// TIA Portal V20 program export: 0 tag tables, 0 data types, 0 data blocks, 4 code blocks (in call order from the OBs), 0 instance data blocks

ORGANIZATION_BLOCK "Main"   // OB1, LAD, ProgramCycle
TITLE = "Main Program Sweep (Cycle)"
{ S7_Optimized_Access := 'TRUE' }
// stored: SetENOAutomatically false
   VAR_INPUT
      Initial_Call : Bool;   // Initial call of this OB
      Remanence : Bool;   // =True, if remanent data are available
   END_VAR
   VAR_TEMP
      unitIndex : SInt;
      query : String;
      paramsTemp : Array[0..5] of Int;
      exec : Bool;
      inWinMC1 : Array[0..1] of Byte;
      outWinMC1 : Array[0..1] of Byte;
      jsonBrand : String;
   END_VAR
BEGIN

REGION Network 1 (SCL): DB_FUNCTION
   //manager database function
   "FC_DBdata"();
   "FC_DBdata2"();
END_REGION

REGION Network 2 (SCL): PLANT
   //manager for plant events
   "DB_plant"();
END_REGION

REGION Network 3 (SCL): WAREHOUSE
   //management of Easybox 1 cycle
   "DB_BOX_1"(Presence_tray1  := "I_OUT_TRAY1",
              Presence_tray2  := "I_OUT_TRAY2",
              Presence_tray3  := "I_OUT_TRAY3",
              Presence_tray4  := "I_OUT_TRAY4",
              Presence_tray5  := "I_OUT_TRAY5",
              Presence_tray6  := "I_OUT_TRAY6",
              Presence_tray7  := "I_OUT_TRAY7",
              Presence_tray8  := "I_OUT_TRAY8",
              Presence_tray9  := "I_OUT_TRAY9",
              Presence_tray10 := "I_OUT_TRAY10",
              Presence_tray11 := "I_OUT_TRAY11",
              Presence_tray12 := "I_OUT_TRAY12",
              // AllTrayInside   := "All_trays_Inside",
              HL_Start_Aux    => "HLStartAux",
              HL_Hold         => "HL_Hold",
              HL_Green        => "HL_GREEN",
              HL_Orange       => "HL_ORANGE",
              HL_Red          => "HL_RED");
END_REGION

REGION Network 4 (SCL): MC1
       // --- ricezione comando cambio brand da HMI (topic TO_PLANT/CMD/BRANDMC1) ---
       IF "DB_MQTT".lastTopicReceived = 'BRANDMC1'
           AND "DB_MQTT".lastCmdReceived >= 1
           AND "DB_MQTT".lastCmdReceived <= 16
       THEN
           "DB_MC1".brandID_req := "DB_MQTT".lastCmdReceived;
           // consumo il comando: evita perdita per dedup di FC_MQTT
           "DB_MQTT".lastCmdReceived := 0;
           "DB_MQTT".lastTopicReceived := '';
       END_IF;

       // --- 0. clamp brandID e latch SOLO a macchina ferma ---
       IF ("DB_MC1".brandID_req < 1) OR ("DB_MC1".brandID_req > 16) THEN
           "DB_MC1".brandID_req := 1;
       END_IF;

       // idle: dispatcher master a 0 (adatta alla tua condizione di "sicuro riconfigurare")
       IF "DB_MC1".Dispatcher[0] = 0 THEN
           "DB_MC1".brandID_act := "DB_MC1".brandID_req;
       END_IF;

       IF ("DB_MC1".brandID_act < 1) OR ("DB_MC1".brandID_act > 16) THEN
           "DB_MC1".brandID_act := 1;
       END_IF;

       // --- 1. finestra ingressi fisici della posizione MC1 ---
       #inWinMC1[0] := "Tag_4";      // byte macchina MC1
       #inWinMC1[1] := 0;          // se il modulo MC1 e' 1 byte lascia 0; se 2 byte: := %IB44;

       // --- 2. mappatura parametrica (config del brand attivo) ---
       "FC_Map_Generic"(inBytes := #inWinMC1,
                        cfg := "DB_MachineConfig".brand["DB_MC1".brandID_act],
                        io_in := "DB_MC1".io_in,
                        io_out := "DB_MC1".io_out,
                        outBytes => #outWinMC1);

       // --- 3. finestra uscite fisiche della posizione MC1 ---
       "Tag_5" := #outWinMC1[0];     // byte uscite macchina MC1
       // se il modulo uscite MC1 e' 2 byte: %QB46 := #outWinMC1[1];

       // --- 4. archetipo di ciclo del brand -> router ---
       "DB_MC1".MachineType := "DB_MachineConfig".brand["DB_MC1".brandID_act].cycleArchetype;

       // --- 5. router (INVARIATO) ---
       "DB_iPos_MC1"(MachineType := "DB_MC1".MachineType,
                     MC_number := 1,
                     MC_inRemoteMode := FALSE,
                     AutoModeFromHandController := NOT "SA_MC1_MANUAL",
                     io_in := "DB_MC1".io_in,
                     io_out := "DB_MC1".io_out,
                     Status := "DB_MC1".Status,
                     Mode := "DB_MC1".Mode,
                     cmd := "DB_MC1".cmd,
                     order := "DB_MC1".order,
                     pallet := "DB_MC1".pallet,
                     fixture := "DB_MC1".fixture,
                     ManualVice := "DB_MC1".ManualVice,
                     piecepresent := "DB_MC1".piecepresent,
                     viceLocked := "DB_MC1".viceLocked,
                     viceUnlocked := "DB_MC1".viceUnlocked,
                     palletLocked := "DB_MC1".palletLocked,
                     changePalletReq := "DB_MC1".changePalletReq,
                     lastMission := "DB_MC1".LastMission,
                     Dispatcher := "DB_MC1".Dispatcher,
                     subState := "DB_MC1".subState,
                     autoModePrev := "DB_MC1".autoModePrev,
                     queryTemp := "DB_MC1".queryTemp,
                     queryStartExecution := "DB_MC1".queryStartExecution);

       // --- pubblica brand attivo (on change) -> FROM_PLANT/BRAND/MC1 ---
       // --- pubblica stato brand (on change di uno qualsiasi dei 4 campi) -> FROM_PLANT/BRAND/MC1 ---
       IF "DB_MC1".brandID_req <> "DB_MC1".brandID_req_old
           OR "DB_MC1".brandID_act <> "DB_MC1".brandID_act_old
           OR "DB_MachineConfig".lastError <> "DB_MC1".cfgErr_old
           OR "DB_MachineConfig".lastErrorBrand <> "DB_MC1".cfgErrBrand_old
       THEN
           #jsonBrand := CONCAT(IN1 := '{"req":',
                                IN2 := "INT_TO_STRING_WITHOUT_SIGN"("DB_MC1".brandID_req),
                                IN3 := ',"act":',
                                IN4 := "INT_TO_STRING_WITHOUT_SIGN"("DB_MC1".brandID_act));
           #jsonBrand := CONCAT(IN1 := #jsonBrand,
                                IN2 := ',"lastError":',
                                IN3 := "INT_TO_STRING_WITHOUT_SIGN"("DB_MachineConfig".lastError),
                                IN4 := ',"lastErrorBrand":',
                                IN5 := "INT_TO_STRING_WITHOUT_SIGN"("DB_MachineConfig".lastErrorBrand),
                                IN6 := '}');
           "FC_MQTT"(insert := true,
                     send := false,
                     topic := 'FROM_PLANT/BRAND/MC1',
                     payload := STRING_TO_WSTRING(#jsonBrand));
           "DB_MC1".brandID_req_old := "DB_MC1".brandID_req;
           "DB_MC1".brandID_act_old := "DB_MC1".brandID_act;
           "DB_MC1".cfgErr_old := "DB_MachineConfig".lastError;
           "DB_MC1".cfgErrBrand_old := "DB_MachineConfig".lastErrorBrand;
       END_IF;
END_REGION

REGION Network 5 (SCL): ROBOT
   //management of >GENERIC< Robot cycle
   "DB_Robot"();

   //read/write infos with robot >SPECIFIC< implementation
   "DB_Robot_Efort"();
END_REGION

REGION Network 6 (SCL): MQTT Comunication

   "LMQTT_Client_DB"(enable := "DB_MQTT".control.enable,
                     publish := "DB_MQTT".control.publish,
                     subscribe := "DB_MQTT".control.subscribe,
                     unsubscribe := "DB_MQTT".control.unsubscribe,
                     qos := "DB_MQTT".qos,
                     retain := "DB_MQTT".retain,
                     publishMsgLen := "DB_MQTT".publishMsgLen,
                     willMsgLen := "DB_MQTT".willMsgLen,
                     timeOut := t#5s,
                     valid => "DB_MQTT".output.valid,
                     done => "DB_MQTT".output.done,
                     busy => "DB_MQTT".output.busy,
                     error => "DB_MQTT".output.error,
                     status => "DB_MQTT".output.status,
                     diagnostics => "DB_MQTT".output.diagnostic,
                     receivedMsgStatus => "DB_MQTT".receiveMsgStatus,
                     receivedMsgDataLen => "DB_MQTT".receivedMsgLen,
                     connParam := "DB_MQTT".connParam,
                     clientIdentifier := "DB_MQTT".clientIdentifier,
                     username := "DB_MQTT".username,
                     password := "DB_MQTT".password,
                     willtopic := "DB_MQTT".willTopic,
                     willMsgPayload := "DB_MQTT".willMsgPayload,
                     mqttTopic := "DB_MQTT".mqttTopic,
                     publishMsgPayload := "DB_MQTT"."publishMsgPayload",
                     receivedTopic := "DB_MQTT".receivedTopic,
                     receivedMsgPayload := "DB_MQTT".receivedMsgPayload);

   "FC_MQTT"(insert := FALSE,
             send := true,
             payload := wstring#'',
             topic := '');
END_REGION

REGION Network 7 (SCL): SQL OPERATION
   // UN SOLO PONTE SQL PER FB7 E FB204 (5/10, ritorno alla configurazione 4-18/9).
   // FB204 e' sul canale 1: il canale 2 resta chiamato a vuoto e non serve nessuno.
   // Precedenza al robot (DB_Robot), FB204 (DB_MC1) passa quando il robot non chiede.
   // Il flag di ciascun richiedente si abbassa SOLO quando la SUA query e' entrata
   // nel ponte; il controllo di lunghezza evita che due stringhe vuote si confermino.

   #query := '';
   #exec := FALSE;
   IF "DB_Robot".queryStartExecution AND LEN("DB_Robot".queryTemp) > 0 THEN
       #query := "DB_Robot".queryTemp;
       #paramsTemp := "DB_Robot".paramsTemp;
       #exec := TRUE;
   ELSIF "DB_MC1".queryStartExecution AND LEN("DB_MC1".queryTemp) > 0 THEN
       #query := "DB_MC1".queryTemp;
       #exec := TRUE;
   END_IF;

   "DB_executeQuery"(query := #query,
                     params := #paramsTemp,
                     exec := #exec);

   IF LEN("DB_Robot".queryTemp) > 0 AND
       "DB_Robot".queryTemp = "SqlCommands".sqlCommands[0] THEN
       "DB_Robot".queryStartExecution := FALSE;
   END_IF;

   IF LEN("DB_MC1".queryTemp) > 0 AND
       "DB_MC1".queryTemp = "SqlCommands".sqlCommands[0] THEN
       "DB_MC1".queryStartExecution := FALSE;
   END_IF;

   // canale 2 chiamato a vuoto: la sorveglianza della connessione resta viva
   "DB_executeQuery2"(query := '',
                      params := #paramsTemp,
                      exec := FALSE);
END_REGION
END_ORGANIZATION_BLOCK

ORGANIZATION_BLOCK "Cyclic interrupt_1"   // OB31, LAD, CyclicInterrupt
{ S7_Optimized_Access := 'TRUE' }
// stored: SetENOAutomatically false
   VAR_INPUT
      Initial_Call : Bool;   // Initial call of this OB
      Event_Count : Int;   // Events discarded
   END_VAR
BEGIN

REGION Network 1 (SCL)
   // "DB_MC2".Status := -1;
END_REGION
END_ORGANIZATION_BLOCK

FUNCTION "FC_DBdata" : Void   // FC2, LAD
{ S7_Optimized_Access := 'TRUE' }
// stored: SetENOAutomatically false
   VAR_TEMP
      tempDataReceived : Bool;   // temp flag for 'dataReceived' from FB 'LSql_Microsoft'
      tempAnalyzeDone : Bool;   // temp flag for 'done' from FB 'AnalyzeTokens'
      tempMetaDataAndRowsAvailable : Bool;   // temp flag for 'metaDataAndRowsAvailable' from FB 'AnalyzeTokens'
      queryTemp : String;
   END_VAR
   VAR_TEMP   // added for the SCL form of the ladder/FBD networks
      _w1 : Bool;
   END_VAR
BEGIN

REGION Network 1 (SCL): nel caso la comunicazione con il DB non parte o cadesse, cerco di ripristinarla dopo un timer
   // Check connection to DB and retry to connect if there is a problem

   "DB_executeQuery".timeoutConnection(IN := "SqlConfig".enableLSql AND "SqlConfig".diagnostics.status > 32770 , //8002
                                       PT := T#2s);

   IF "DB_executeQuery".timeoutConnection.Q THEN
       "SqlConfig".enableLSql := false;
   END_IF;

   "DB_executeQuery".timeoutRetrayConnection(IN := NOT "SqlConfig".enableLSql,
                                             PT := T#1s);

   IF "DB_executeQuery".timeoutRetrayConnection.Q THEN
       "SqlConfig".enableLSql := true;
   END_IF;
END_REGION

REGION Network 2: TDS Connection and Communication Handling
   // this network handles the TDS connection and communication
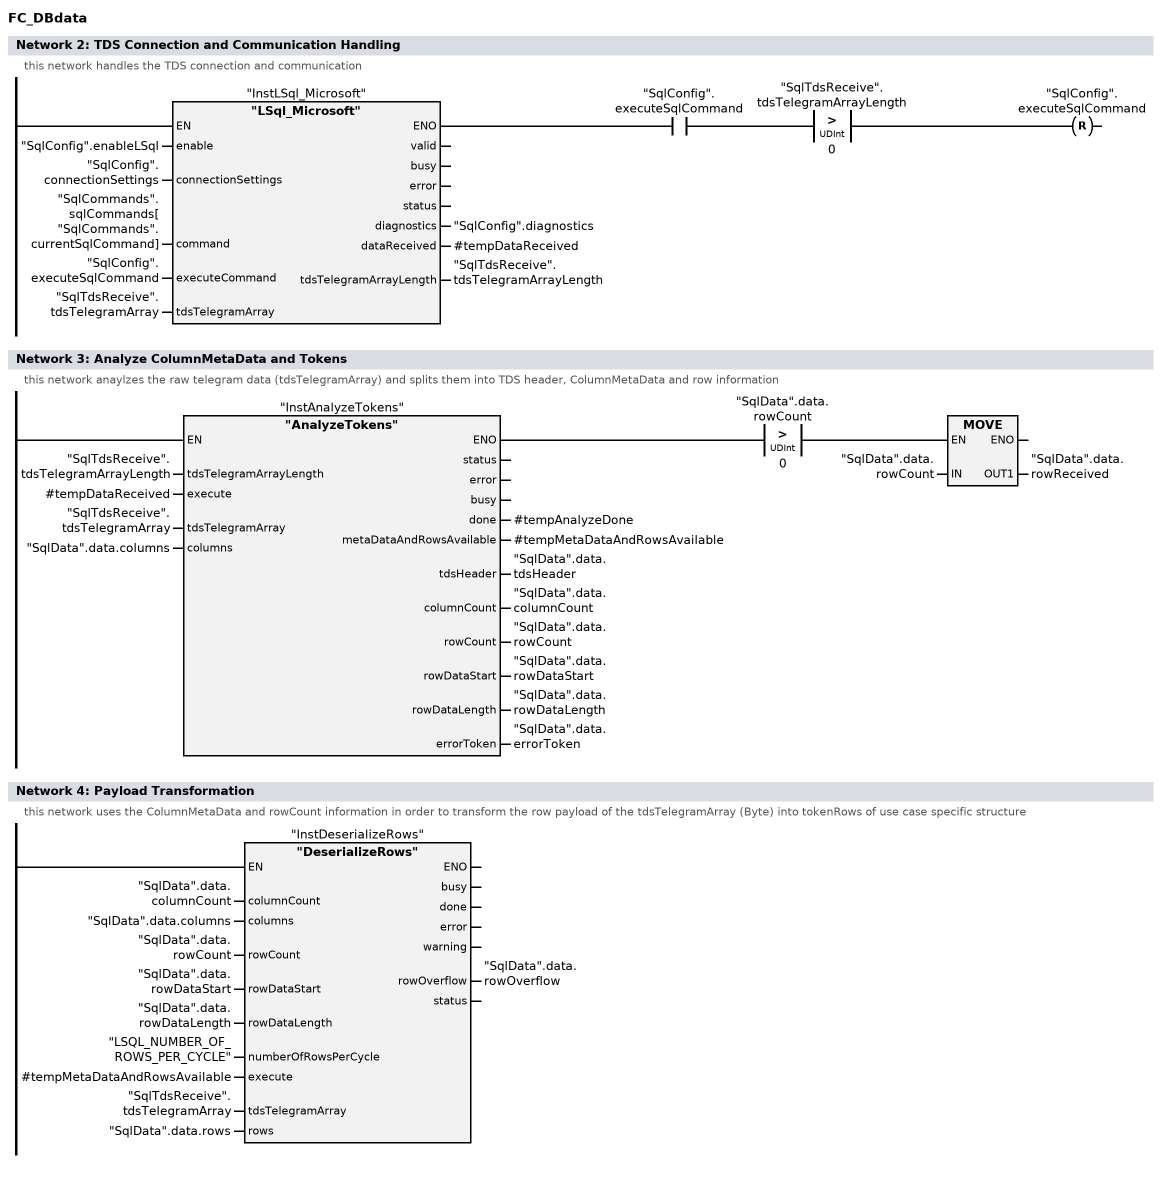
   RUNG wire#powerrail
      "InstLSql_Microsoft"(enable := "SqlConfig".enableLSql, connectionSettings := "SqlConfig".connectionSettings, command := "SqlCommands".sqlCommands["SqlCommands".currentSqlCommand], executeCommand := "SqlConfig".executeSqlCommand, tdsTelegramArray := "SqlTdsReceive".tdsTelegramArray, valid =>, busy =>, error =>, status =>, diagnostics => "SqlConfig".diagnostics, dataReceived => #tempDataReceived, tdsTelegramArrayLength => "SqlTdsReceive".tdsTelegramArrayLength)
      Contact( "SqlConfig".executeSqlCommand )
      { S7_Templates := "SrcType := UDInt" } GT_Contact(in1 := "SqlTdsReceive".tdsTelegramArrayLength, in2 := 0)
      R_Coil( "SqlConfig".executeSqlCommand )
   END_RUNG
   // the same network as SCL:
   "InstLSql_Microsoft"(enable := "SqlConfig".enableLSql,   // "LSql_Microsoft"
                        connectionSettings := "SqlConfig".connectionSettings,
                        command := "SqlCommands".sqlCommands["SqlCommands".currentSqlCommand],
                        executeCommand := "SqlConfig".executeSqlCommand,
                        tdsTelegramArray := "SqlTdsReceive".tdsTelegramArray,
                        diagnostics => "SqlConfig".diagnostics,
                        dataReceived => #tempDataReceived,
                        tdsTelegramArrayLength => "SqlTdsReceive".tdsTelegramArrayLength,
                        ENO => #_w1);
   IF #_w1 AND "SqlConfig".executeSqlCommand AND ("SqlTdsReceive".tdsTelegramArrayLength > 0) THEN
       "SqlConfig".executeSqlCommand := FALSE;
   END_IF;
END_REGION

REGION Network 3: Analyze ColumnMetaData and Tokens
   // this network anaylzes the raw telegram data (tdsTelegramArray) and splits them into TDS header, ColumnMetaData and row information
   RUNG wire#powerrail
      "InstAnalyzeTokens"(tdsTelegramArrayLength := "SqlTdsReceive".tdsTelegramArrayLength, execute := #tempDataReceived, tdsTelegramArray := "SqlTdsReceive".tdsTelegramArray, columns := "SqlData".data.columns, status =>, error =>, busy =>, done => #tempAnalyzeDone, metaDataAndRowsAvailable => #tempMetaDataAndRowsAvailable, tdsHeader => "SqlData".data.tdsHeader, columnCount => "SqlData".data.columnCount, rowCount => "SqlData".data.rowCount, rowDataStart => "SqlData".data.rowDataStart, rowDataLength => "SqlData".data.rowDataLength, errorToken => "SqlData".data.errorToken)
      { S7_Templates := "SrcType := UDInt" } GT_Contact(in1 := "SqlData".data.rowCount, in2 := 0)
      Move(in := "SqlData".data.rowCount, out1 => "SqlData".data.rowReceived)
   END_RUNG
   // the same network as SCL:
   "InstAnalyzeTokens"(tdsTelegramArrayLength := "SqlTdsReceive".tdsTelegramArrayLength,   // "AnalyzeTokens"
                       execute := #tempDataReceived,
                       tdsTelegramArray := "SqlTdsReceive".tdsTelegramArray,
                       columns := "SqlData".data.columns,
                       done => #tempAnalyzeDone,
                       metaDataAndRowsAvailable => #tempMetaDataAndRowsAvailable,
                       tdsHeader => "SqlData".data.tdsHeader,
                       columnCount => "SqlData".data.columnCount,
                       rowCount => "SqlData".data.rowCount,
                       rowDataStart => "SqlData".data.rowDataStart,
                       rowDataLength => "SqlData".data.rowDataLength,
                       errorToken => "SqlData".data.errorToken,
                       ENO => #_w1);
   IF #_w1 AND ("SqlData".data.rowCount > 0) THEN
       "SqlData".data.rowReceived := "SqlData".data.rowCount;
   END_IF;
END_REGION

REGION Network 4: Payload Transformation
   // this network uses the ColumnMetaData and rowCount information in order to transform the row payload of the tdsTelegramArray (Byte) into tokenRows of use case specific structure
   RUNG wire#powerrail
      "InstDeserializeRows"(columnCount := "SqlData".data.columnCount, columns := "SqlData".data.columns, rowCount := "SqlData".data.rowCount, rowDataStart := "SqlData".data.rowDataStart, rowDataLength := "SqlData".data.rowDataLength, numberOfRowsPerCycle := "LSQL_NUMBER_OF_ROWS_PER_CYCLE", execute := #tempMetaDataAndRowsAvailable, tdsTelegramArray := "SqlTdsReceive".tdsTelegramArray, rows := "SqlData".data.rows, busy =>, done =>, error =>, warning =>, rowOverflow => "SqlData".data.rowOverflow, status =>)
   END_RUNG
   // the same network as SCL:
   "InstDeserializeRows"(columnCount := "SqlData".data.columnCount,   // "DeserializeRows"
                         columns := "SqlData".data.columns,
                         rowCount := "SqlData".data.rowCount,
                         rowDataStart := "SqlData".data.rowDataStart,
                         rowDataLength := "SqlData".data.rowDataLength,
                         numberOfRowsPerCycle := "LSQL_NUMBER_OF_ROWS_PER_CYCLE",
                         execute := #tempMetaDataAndRowsAvailable,
                         tdsTelegramArray := "SqlTdsReceive".tdsTelegramArray,
                         rows := "SqlData".data.rows,
                         rowOverflow => "SqlData".data.rowOverflow);
END_REGION
END_FUNCTION

FUNCTION "FC_ExtractGripper" : Void   // FC9, LAD
{ S7_Optimized_Access := 'TRUE' }
// stored: SetENOAutomatically false
   VAR_INPUT
      GripperVal : DInt;
   END_VAR
   VAR_OUTPUT
      Gripper1 : Int;
      Gripper2 : Int;
   END_VAR
BEGIN

REGION Network 1 (SCL)
   IF #GripperVal < 1000 THEN
       #Gripper1 := DINT_TO_INT(#GripperVal);
       #Gripper2 := 0;
   ELSE
       #Gripper1 := TRUNC_INT(#GripperVal / 1000);
       #Gripper2 := DINT_TO_INT(#GripperVal ) - (TRUNC_INT(#GripperVal / 1000) * 1000);
   END_IF;
END_REGION
END_FUNCTION
